FUNCTION_BLOCK fbMachineCycleCounter	//Blok funkcyjny wykorzystywany do obliczenia przebiegu maszyny
VAR_INPUT
	stTimeStruct		: stAircomTimeStruct;
	iMaximalOperations	: ULINT := 100000;
END_VAR
VAR_OUTPUT
	iMakedOperations	: ULINT;
	iMakedCycles		: ULINT;
END_VAR
VAR PERSISTENT
	iOperationCalc		: ULINT;	//Liczba wykonanych operacji
	iCyclesCalc			: ULINT;	//Liczba wykonanych produktów
	bError				: BOOL;
	bWarning			: BOOL;
	arWarningTable		: ARRAY[0..10] OF ULINT;
	arResetHistory		: ARRAY[0..100] OF stResetHistory;
END_VAR
VAR
	fbShiftFilter		: R_TRIG;
	fbErrorOccur		: R_TRIG;
	fbWarningTrigger	: R_TRIG;
	bBlocked			: BOOL;
	sUserName			: STRING;
	bResetAqusitton		: BOOL := TRUE;
	bTempolaryPermit	: BOOL := TRUE;
	bClear				: BOOL;
	bReset				: BOOL;
	iOperationCalcHMI	: UDINT;
	iCyclesCalcHMI		: UDINT;
END_VAR

//New shift reader
fbShiftFilter(CLK:=stTimeStruct.bNew_Shift);
fbErrorOccur(CLK:=(iOperationCalc >= iMaximalOperations));
fbWarningTrigger(CLK:=tWarningTrigger);

pError 		S= (fbShiftFilter.Q AND iOperationCalc >= iMaximalOperations) OR fbErrorOccur.Q;
pWarning	S= fbWarningTrigger.Q;

iMakedOperations 	:= iOperationCalc;
iMakedCycles		:= iCyclesCalc;
iOperationCalcHMI	:= ULINT_TO_UDINT(iOperationCalc);
iCyclesCalcHMI		:= ULINT_TO_UDINT(iCyclesCalc);

bBlocked := (GVL.fbUserLogin.sUserName <> '' AND GVL.fbUserLogin.sUserName <> 'Maintenance User') AND GVL.fbUserLogin.bUserLogged;

sUserName	:= GVL.fbUserLogin.sUserName;

IF bClear THEN
	mResetError(sWorkerID := sUserName);
	bClear := FALSE;
END_IF

IF bReset THEN
	mResetOperaionCalc(sWorkerID := sUserName);
	bReset := FALSE;
END_IF

METHOD mCalcCycle : BOOL
VAR_INPUT
END_VAR
iCyclesCalc := iCyclesCalc + 1;
mCalcCycle := TRUE;
END_METHOD

METHOD mCalcOperation : BOOL
VAR_INPUT
END_VAR
iOperationCalc := iOperationCalc + 1;
mCalcOperation := TRUE;
END_METHOD

METHOD mResetError : BOOL
VAR_INPUT
	sWorkerID		: STRING;
END_VAR
VAR
	iBuffer			: UINT;
END_VAR
FOR iBuffer := 0 TO 100 DO
	IF arResetHistory[iBuffer].iOperationAmout = 0 THEN
		arResetHistory[iBuffer].iCyclesAmount			:= iCyclesCalc;
		arResetHistory[iBuffer].iOperationAmout			:= iOperationCalc;
		arResetHistory[iBuffer].sOperationDescription	:= 'Reseting Error By To Much Of Operations';
		arResetHistory[iBuffer].stDate					:= stTimeStruct;
		arResetHistory[iBuffer].sWorkerID				:= sWorkerID;
		pError := FALSE;
		IF iBuffer < 100 THEN
			MEMSET(destAddr:=ADR(arResetHistory[iBuffer + 1]),fillByte:= 0,n:=SIZEOF(arResetHistory[iBuffer + 1]));
		ELSE
			MEMSET(destAddr:=ADR(arResetHistory[0]),fillByte:= 0,n:=SIZEOF(arResetHistory[0]));	
		END_IF
		EXIT;
	END_IF
END_FOR
END_METHOD

METHOD mResetOperaionCalc : BOOL
VAR_INPUT
	sWorkerID		: STRING;
END_VAR
VAR
	iBuffer			: UINT;
END_VAR

//Add record to history
FOR iBuffer := 0 TO 100 DO
	IF arResetHistory[iBuffer].iOperationAmout = 0 THEN
		arResetHistory[iBuffer].iCyclesAmount			:= iCyclesCalc;
		arResetHistory[iBuffer].iOperationAmout			:= iOperationCalc;
		arResetHistory[iBuffer].sOperationDescription	:= 'Reseting Number Of Operations';
		arResetHistory[iBuffer].stDate					:= stTimeStruct;
		arResetHistory[iBuffer].sWorkerID				:= sWorkerID;
		iOperationCalc := 0;
		IF iBuffer < 100 THEN
			MEMSET(destAddr:=ADR(arResetHistory[iBuffer + 1]),fillByte:= 0,n:=SIZEOF(arResetHistory[iBuffer + 1]));
		ELSE
			MEMSET(destAddr:=ADR(arResetHistory[0]),fillByte:= 0,n:=SIZEOF(arResetHistory[0]));	
		END_IF
		EXIT;
	END_IF
END_FOR
mResetOperaionCalc := (iOperationCalc = 0);
END_METHOD

METHOD mResetWarning : BOOL
VAR_INPUT
END_VAR
pWarning := FALSE;
mResetWarning := TRUE;
END_METHOD

PROPERTY pError : BOOL
GET
pError	:= bError;
END_GET
SET
bError	:= pError;
END_SET
END_PROPERTY

PROPERTY pWarning : BOOL
GET
pWarning	:= bWarning;
END_GET
SET
bWarning := pWarning;
END_SET
END_PROPERTY

TRANSITION tWarningTrigger:
tWarningTrigger := 
	((arWarningTable[0] = iOperationCalc) AND (arWarningTable[0] <> 0)) OR ((arWarningTable[1] = iOperationCalc) AND (arWarningTable[1] <> 0)) OR ((arWarningTable[2] = iOperationCalc) AND (arWarningTable[2] <> 0)) OR
	((arWarningTable[3] = iOperationCalc) AND (arWarningTable[3] <> 0)) OR ((arWarningTable[4] = iOperationCalc) AND (arWarningTable[4] <> 0)) OR ((arWarningTable[5] = iOperationCalc) AND (arWarningTable[5] <> 0)) OR
	((arWarningTable[6] = iOperationCalc) AND (arWarningTable[6] <> 0)) OR ((arWarningTable[7] = iOperationCalc) AND (arWarningTable[7] <> 0)) OR ((arWarningTable[8] = iOperationCalc) AND (arWarningTable[8] <> 0)) OR
	((arWarningTable[9] = iOperationCalc) AND (arWarningTable[9] <> 0)) OR ((arWarningTable[10] = iOperationCalc) AND (arWarningTable[10] <> 0));
END_TRANSITION

END_FUNCTION_BLOCK

(* stored: Version 1.1.0.1, ProductVersion 3.1.4024.13
   POU fbMachineCycleCounter: Id {f86b8b51-6646-066d-3532-ee0c4e6b970b}, SpecialFunc None
   Method mCalcCycle: Id {a3a75e60-2570-0415-09bc-e8ca0843042a}
   Method mCalcOperation: Id {df70b1d5-555d-05a8-163f-c116232ccdc7}
   Method mResetError: Id {27816e82-9c72-0dcd-1865-0e4977b8f917}
   Method mResetOperaionCalc: Id {7e9c204d-87a8-0752-3c35-99fc14080479}
   Method mResetWarning: Id {0f5c8030-f7c4-0335-1868-083b4db1220f}
   Property pError: Id {6e2b6988-54b0-08ee-2417-556729a1442c}
   Get Get: Id {36e29819-211c-06ba-2b20-a27d716c494b}
   Set Set: Id {e3a97019-f62a-0e9b-0a8c-00b947aa84b1}
   Property pWarning: Id {1648e1a8-e65b-03f4-0f8c-d07fcd89081f}
   Get Get: Id {6d5c552c-034b-0939-3e18-92d3bffe812b}
   Set Set: Id {0e06ce6b-32ed-0e32-20e8-a6bb683645e1}
   Transition tWarningTrigger: Id {67cbd215-2c2f-0d5f-2ebe-bf06970f33b8} *)
